FUNCTION_BLOCK F_DEAD_ZONE2 (* Basic Function Block Type *)
  (* Standard: 61499-2; Classification: Control Modules; Description: DEAD_ZONE is a linear transfer function with dead zone. The output equals the input signal when the absolute value of the input is greater than L. DEAD_ZONE = X if ABS(X) > L DEAD_ZONE = 0 if ABS(X) <= L *)
  (* Version 0.0, 2011-08-27, 4DIAC-IDE, 4DIAC-Consortium *)
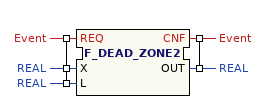
  EVENT_INPUT
    REQ WITH X, L; (* Normal Execution Request *)
  END_EVENT
  EVENT_OUTPUT
    CNF WITH OUT; (* Execution Confirmation *)
  END_EVENT
  VAR_INPUT
    X : REAL; (* input *)
    L : REAL; (* lockout value *)
  END_VAR
  VAR_OUTPUT
    OUT : REAL; (* output value *)
  END_VAR
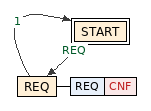
  EC_STATES
    START; (* Initial State *)
    REQ : REQ -> CNF; (* Normal execution *)
  END_STATES
  EC_TRANSITIONS
    START TO REQ := REQ;
    REQ TO START := 1;
  END_TRANSITIONS
  ALGORITHM REQ IN ST: (* Normally executed algorithm *)
IF ABS(X) > L THEN
	OUT := X;
ELSIF OUT > 0.0 THEN
	OUT := L;
ELSE
	OUT := -L;
END_IF;
  END_ALGORITHM
END_FUNCTION_BLOCK
